TYPE ST_PeakShaveBox_Get :
STRUCT
	PSBmode				: ePSBMode;
	Powermonitor 		: st_MeasurementVoltageData;
	PowerStatus			: st_PowerMeasurement_status;
	r_MaxCTCurrent		: REAL:= 4000;
	b_buscouplerReady	: BOOL;
	b_active			: BOOL;
	b_dataOK			: BOOL;
	b_ContactorFb		: BOOL;
	b_SyncFb			: BOOL;
	b_SettingsChangePending	:	BOOL;
END_STRUCT
END_TYPE

(* stored: Version 1.1.0.1, ProductVersion 3.1.4024.12
   DUT ST_PeakShaveBox_Get: Id {33c5722f-15da-4d92-854e-828c06ec61ce} *)
